SUBAPPLICATION Uebung_152_AX (* Impulszähler & PI Regler, mit Plug and Socket (Adapter-Native) *)
  (* Standard: 61499-2; Description: Copyright (c) 2026 Meisterschulen am Ostbahnhof This program and the accompanying materials are made available under the terms of the Eclipse Public License 2.0 which is available at https://www.eclipse.org/legal/epl-2.0/ SPDX-License-Identifier: EPL-2.0 *)
  (* Version 1.3, 2026-10-03, Franz Höpfinger, Meisterschulen am Ostbahnhof, Folgefix zu CTRL_PI_AR v1.3 (SUP/OFS/LL/LH jetzt AR-Adapter-Sockets) und FT_DERIV_10_AR v1.2 (K jetzt AUI-Adapter-Socket): bisherige Parameter SUP/OFS/M_I/KP/KI/LL/LH auf CTRL_PI und K auf FT_DERIV entfernt (waeren jetzt IDE-Fehler, da keine plain InputVars mehr) - durch initval_AR/initval_AUI-Literale + AdapterConnections ersetzt, gleiche Werte wie bisher. M_I/KP/KI waren schon seit v1.1 (CTRL_PI_AR-Umstellung auf Adapter) als Parameter falsch verdrahtet (nie korrigiert), jetzt mitgefixt. *)
  (* Version 1.2, 2026-09-15, Franz Höpfinger, Meisterschulen am Ostbahnhof, SET-Eingang an CTRL_PI auf AR-Adapter (initval_AR) umgestellt. *)
  (* Version 1.1, 2026-09-12, Franz Höpfinger, Meisterschulen am Ostbahnhof, Vollstaendig auf Adapter-Architektur umgestellt: FT_DERIV_10_AR und CTRL_PI_AR aus OSCAT_adapter, AD_TO_AR_NUM und AR_TO_AD_NUM fuer sauberen Adapterdatenfluss. *)
  (* Version 1.0, 2026-09-10, Franz Höpfinger, Meisterschulen am Ostbahnhof, initial API and implementation and/or initial documentation *)
  PACKAGE Uebungen;
  IMPORT logiBUS::io::DI::logiBUS_DI::Input_I1;
  IMPORT logiBUS::io::DI::logiBUS_DI::Input_I2;
  IMPORT logiBUS::io::DI::logiBUS_DI::Input_I3;
  IMPORT logiBUS::io::DI::logiBUS_DI_Events::BUTTON_SINGLE_CLICK;
  IMPORT logiBUS::io::DQ::logiBUS_DO::Output_Q1;
  IMPORT logiBUS::io::PI::logiBUS_PI::PulseInput_I8;
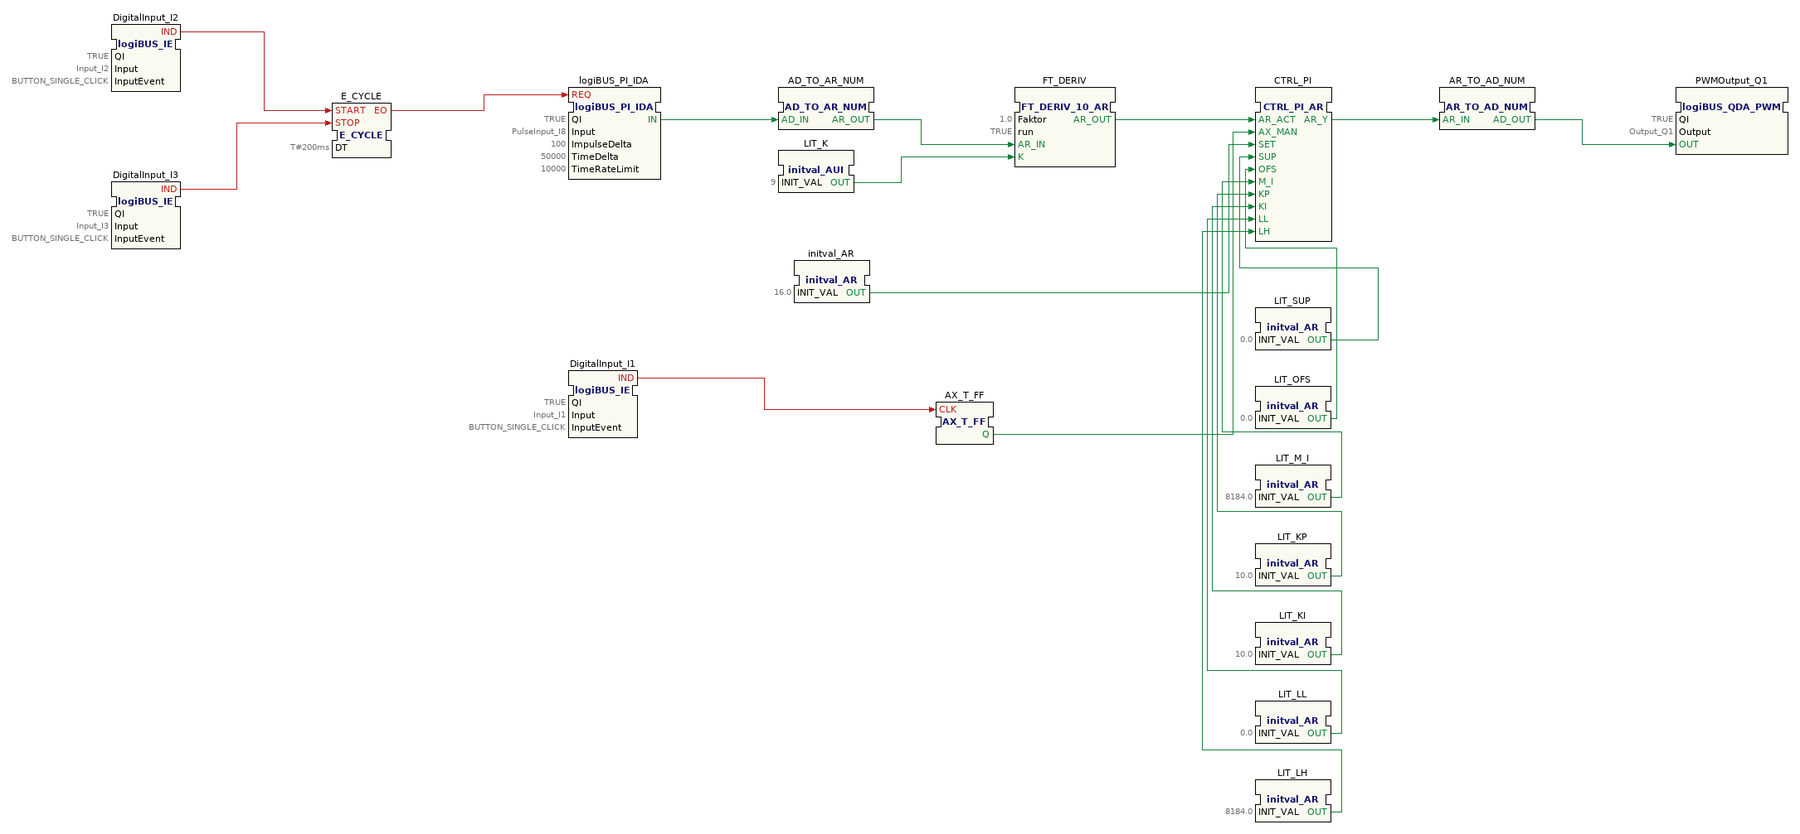
  FBS
    DigitalInput_I2 : logiBUS::io::DI::logiBUS_IE(QI := TRUE, Input := Input_I2, InputEvent := BUTTON_SINGLE_CLICK);
    DigitalInput_I3 : logiBUS::io::DI::logiBUS_IE(QI := TRUE, Input := Input_I3, InputEvent := BUTTON_SINGLE_CLICK);
    E_CYCLE : iec61499::events::E_CYCLE(DT := T#200ms);
    logiBUS_PI_IDA : logiBUS::io::PI::logiBUS_PI_IDA(QI := TRUE, Input := PulseInput_I8, ImpulseDelta := 100, TimeDelta := 50000, TimeRateLimit := 10000);
    AD_TO_AR_NUM : adapter::conversion::unidirectional::AD_TO_AR_NUM;
    FT_DERIV : OSCAT_adapter::Control::FT_DERIV_10_AR(Faktor := 1.0, run := TRUE);
    LIT_K : adapter::types::unidirectional::AUI::initval::initval_AUI(INIT_VAL := 9);
    DigitalInput_I1 : logiBUS::io::DI::logiBUS_IE(QI := TRUE, Input := Input_I1, InputEvent := BUTTON_SINGLE_CLICK);
    AX_T_FF : adapter::events::unidirectional::AX_T_FF;
    CTRL_PI : OSCAT_adapter::Control::CTRL_PI_AR;
    LIT_SUP : adapter::types::unidirectional::AR::initval::initval_AR(INIT_VAL := 0.0);
    LIT_OFS : adapter::types::unidirectional::AR::initval::initval_AR(INIT_VAL := 0.0);
    LIT_M_I : adapter::types::unidirectional::AR::initval::initval_AR(INIT_VAL := 8184.0);
    LIT_KP : adapter::types::unidirectional::AR::initval::initval_AR(INIT_VAL := 10.0);
    LIT_KI : adapter::types::unidirectional::AR::initval::initval_AR(INIT_VAL := 10.0);
    LIT_LL : adapter::types::unidirectional::AR::initval::initval_AR(INIT_VAL := 0.0);
    LIT_LH : adapter::types::unidirectional::AR::initval::initval_AR(INIT_VAL := 8184.0);
    AR_TO_AD_NUM : adapter::conversion::unidirectional::AR_TO_AD_NUM;
    PWMOutput_Q1 : logiBUS::io::DQ::logiBUS_QDA_PWM(QI := TRUE, Output := Output_Q1);
    initval_AR : adapter::types::unidirectional::AR::initval::initval_AR(INIT_VAL := 16.0);
  END_FBS
  EVENT_CONNECTIONS
    DigitalInput_I2.IND TO E_CYCLE.START;
    DigitalInput_I3.IND TO E_CYCLE.STOP;
    E_CYCLE.EO TO logiBUS_PI_IDA.REQ;
    DigitalInput_I1.IND TO AX_T_FF.CLK;
  END_CONNECTIONS
  ADAPTER_CONNECTIONS
    logiBUS_PI_IDA.IN TO AD_TO_AR_NUM.AD_IN;
    AD_TO_AR_NUM.AR_OUT TO FT_DERIV.AR_IN;
    LIT_K.OUT TO FT_DERIV.K;
    FT_DERIV.AR_OUT TO CTRL_PI.AR_ACT;
    AX_T_FF.Q TO CTRL_PI.AX_MAN;
    CTRL_PI.AR_Y TO AR_TO_AD_NUM.AR_IN;
    AR_TO_AD_NUM.AD_OUT TO PWMOutput_Q1.OUT;
    initval_AR.OUT TO CTRL_PI.SET;
    LIT_SUP.OUT TO CTRL_PI.SUP;
    LIT_OFS.OUT TO CTRL_PI.OFS;
    LIT_M_I.OUT TO CTRL_PI.M_I;
    LIT_KP.OUT TO CTRL_PI.KP;
    LIT_KI.OUT TO CTRL_PI.KI;
    LIT_LL.OUT TO CTRL_PI.LL;
    LIT_LH.OUT TO CTRL_PI.LH;
  END_CONNECTIONS
END_SUBAPPLICATION
